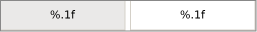
VISUALIZATION VISU_ConfigLREAL1Entry  // 257x32
VAR_IN_OUT
    active : LREAL;
    editable : LREAL;
END_VAR
    Textfield (0,0 125x30), "%.1f", text variable: active, input disabled if: TRUE
    Textfield (130,0 125x30), "%.1f", text variable: editable, colour toggle: editable <> active
        OnMouseClick: write the text variable via Default
END_VISUALIZATION

(* stored: Version 1.1.0.1, ProductVersion 3.1.0.36
   Visu VISU_ConfigLREAL1Entry: Id {29ec5ceb-2bc2-4d29-9315-b1a24192a47d} *)
